GLOBALCONSTANTS anlagenSequenz (* Global constants für AnlagenSequenz_06 (STATUS_BETRIEB/STATUS_STOERUNG), s. KONZEPT_Anlagensequenz.md *)
  (* Standard: 61499-1; Description: Copyright (c) 2026 HR Agrartechnik GmbH This program and the accompanying materials are made available under the terms of the Eclipse Public License 2.0 which is available at https://www.eclipse.org/legal/epl-2.0/ SPDX-License-Identifier: EPL-2.0 *)
  (* Version 1.0, 2026-08-12, Franz Höpfinger, HR Agrartechnik GmbH *)
  PACKAGE logiBUS::utils::sequence::const;
  VAR_GLOBAL CONSTANT
    STATUS_BETRIEB_AUS : SINT := SINT#0; (* Anlage steht *)
    STATUS_BETRIEB_HOCHFAHREN : SINT := SINT#1; (* Vorlauf-Kette aktiv *)
    STATUS_BETRIEB_LAEUFT : SINT := SINT#2; (* alle 6 Motoren laufen *)
    STATUS_BETRIEB_HERUNTERFAHREN : SINT := SINT#3; (* Nachlauf-Kette aktiv *)
    STATUS_STOERUNG_KEINE : SINT := SINT#0; (* keine aktive Störung *)
    STATUS_STOERUNG_AKTIV : SINT := SINT#4; (* Störung aktiv, verriegelt bis EIN *)
    TRANSIT_ART_KEINE : SINT := SINT#0; (* kein Motor aktuell im Vor-/Nachlauf (S_AUS, S_LAEUFT) *)
    TRANSIT_ART_VORLAUF : SINT := SINT#1; (* TRANSIT_MOTOR startet nach Ablauf der aktuellen Zeit *)
    TRANSIT_ART_NACHLAUF : SINT := SINT#2; (* TRANSIT_MOTOR stoppt nach Ablauf der aktuellen Zeit *)
  END_VAR
END_GLOBALCONSTANTS
